//{attribute 'qualified_only'}
{attribute 'strict'}
TYPE eMarking_Types :
(
		Plain_Text 		:= 0 ,
		DataMatrix_2D 	:= 1 ,
		QR_Code 		:= 2 ,
		BarCode 		:= 3 
);
END_TYPE

(* stored: Version 1.1.0.1, ProductVersion 3.1.4024.3
   EnumerationTextList eMarking_Types: Id {b18ef9d7-c93a-4f44-8362-84317daea5c1} *)
